TYPE Basic_MC_Power_Status_typ : 	
	STRUCT 
		Status : BOOL;
		Busy : BOOL;
	END_STRUCT
END_TYPE

(* stored: Version 1.1.0.1, ProductVersion 3.1.4024.3
   DUT Basic_MC_Power_Status_typ: Id {bddee05b-d25e-0272-1531-7894352f6008} *)
